// TIA Portal V21 export
TYPE "LAxisCtrl_typePhasing"
TITLE = LAxisCtrl_typePhasing
// Support: tech.team.motioncontrol@siemens.com
   STRUCT
      phaseShift : LReal := 0.0;   // Absolute or relative leading value shift
      velocity : LReal := -1.0;   // Velocity for leading value shift, added to synchronous operation motion (Value > 0.0: The specified value is used; Value = 0.0: Not permitted; Value < 0.0: Use of the default value configured in the technology object)
      acceleration : LReal := -1.0;   // Acceleration for leading value shift, added to synchronous operation motion (Value > 0.0: The specified value is used; Value = 0.0: Not permitted; Value < 0.0: Use of the default value configured in the technology object)
      deceleration : LReal := -1.0;   // Deceleration for leading value shift, added to synchronous operation motion (Value > 0.0: The specified value is used; Value = 0.0: Not permitted; Value < 0.0: Use of the default value configured in the technology object)
      jerk : LReal := -1.0;   // Jerk for leading value shift, added to synchronous operation motion (Value > 0.0: Smooth velocity profile, the specified value is used; Value = 0.0: Trapezoid velocity profile; Value < 0.0: Use of the default value configured in the technology object)
      profileReference : DInt;   // Type of traversing of the leading value offset (0: Only with gearing: Traverse leading value offset using dynamics parameters; 1: Traverse leading value offset via leading value distance starting from current leading value position; 2: Traverse leading value offset from leading value position "StartPosition"; 5: Cancel only one waiting job for the leading value offset)
      phasingDistance : LReal;   // Leading value distance (Distance of the leading axis during the traversing of the leading value offset) when "ProfileReference" = 1, 2
      startPosition : LReal;   // Leading value position starting from which the leading value offset is traversed when "ProfileReference" = 2
      direction : DInt := 3;   // Direction of the leading value distance (1: Positive direction; 2: Negative direction; 3: Current direction) when "ProfileReference" = 1, 2
      phaseAbsolute : Bool := TRUE;   // Indicates the type of phase shift. TRUE: Shift the leading value as an absolute shift; FALSE: Shift the leading value relative to the existing leading value shift
      phaseShiftChangeOnTheFly : Bool := FALSE;   // TRUE: Changing phase shift on-the-fly at absolute phasing; FALSE: Phase shift change requires a new rising edge at phasing input
   END_STRUCT;
END_TYPE
